(* Logix 5000 project; controller GEA_Test_Chamber vendor 1 type 14 code 196 rev 32.14; software revision 32.04; part 7 of 11 *)
(* tags used below, declared in another part *)
   FVIR_1_S_Step : INT;
   FVIR_1_W_Step : INT;
   FVIR_2_S_Step : INT;
   FVIR_2_W_Step : INT;
   FVIR_3_S_Step : INT;
   FVIR_3_W_Step : INT;
   FVIR_4_S_Step : INT;
   FVIR_4_W_Step : INT;
   FVIR_LabView_Comm_OK : BOOL;
   Start_Manequinn_Seq : BOOL;
   Start_Spill_Gasoline : BOOL;
   Start_Water_Flow_T1S : BOOL;
   Start_Water_Flow_T1W : BOOL;
   Start_Water_Flow_T2S : BOOL;
   Start_Water_Flow_T2W : BOOL;
   Start_Water_Flow_T3S : BOOL;
   Start_Water_Flow_T3W : BOOL;
   Start_Water_Flow_T4S : BOOL;
   Start_Water_Flow_T4W : BOOL;
   test : BOOL;
   Timer_Delay : TIMER[30];
   FVIR_LabView_Control : INT;
   FVIR_Test_No : INT;
   Output_FVIR : Output_FVIR;
   SET_0 : BOOL;
(* FVIR_Chamber, continued *)

ROUTINE FVIR_Test_1_Summer   (* ladder *)
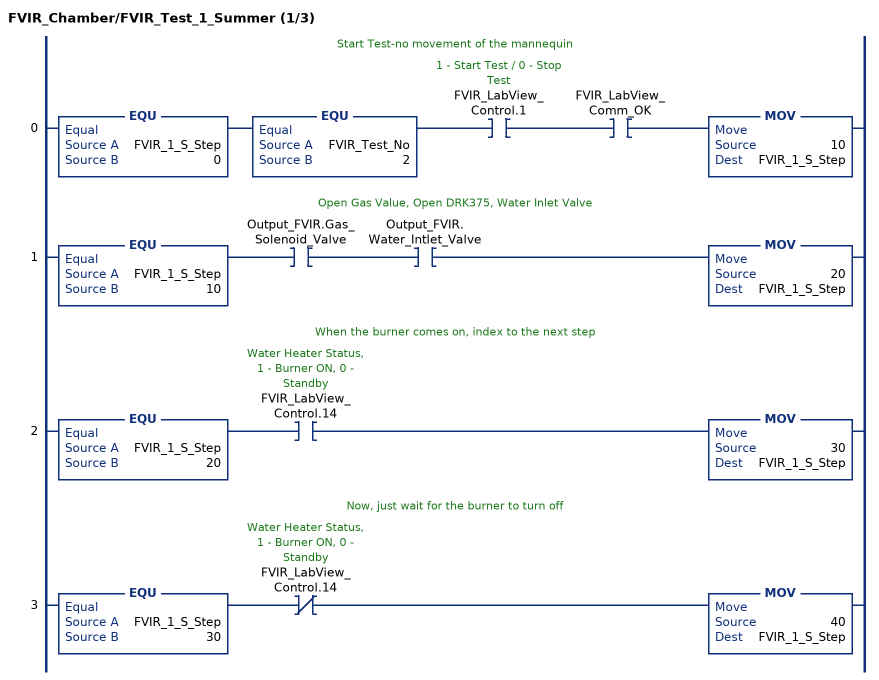
   // Start Test-no movement of the mannequin
   0: EQU(FVIR_1_S_Step,0)EQU(FVIR_Test_No,2)XIC(FVIR_LabView_Control.1)XIC(FVIR_LabView_Comm_OK)MOV(10,FVIR_1_S_Step);
   // Open Gas Value, Open DRK375, Water Inlet Valve
   1: EQU(FVIR_1_S_Step,10)XIC(Output_FVIR.Gas_Solenoid_Valve)XIC(Output_FVIR.Water_Intlet_Valve)MOV(20,FVIR_1_S_Step);
   // When the burner comes on, index to the next step
   2: EQU(FVIR_1_S_Step,20)XIC(FVIR_LabView_Control.14)MOV(30,FVIR_1_S_Step);
   // Now, just wait for the burner to turn off
   3: EQU(FVIR_1_S_Step,30)XIO(FVIR_LabView_Control.14)MOV(40,FVIR_1_S_Step);
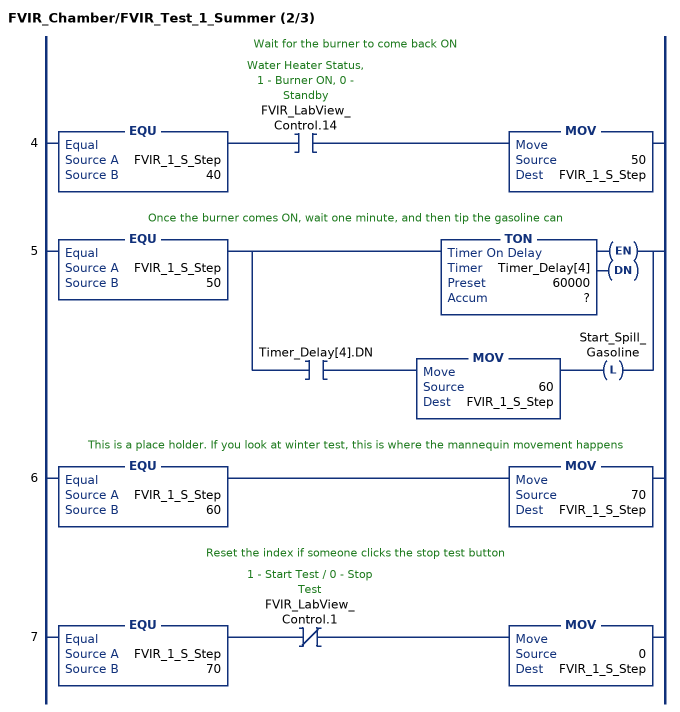
   // Wait for the burner to come back ON
   4: EQU(FVIR_1_S_Step,40)XIC(FVIR_LabView_Control.14)MOV(50,FVIR_1_S_Step);
   // Once the burner comes ON, wait one minute, and then tip the gasoline can
   5: EQU(FVIR_1_S_Step,50)[TON(Timer_Delay[4],?,?) ,XIC(Timer_Delay[4].DN) MOV(60,FVIR_1_S_Step) OTL(Start_Spill_Gasoline) ];
   // This is a place holder. If you look at winter test, this is where the mannequin movement happens
   6: EQU(FVIR_1_S_Step,60)MOV(70,FVIR_1_S_Step);
   // Reset the index if someone clicks the stop test button
   7: EQU(FVIR_1_S_Step,70)XIO(FVIR_LabView_Control.1)MOV(0,FVIR_1_S_Step);
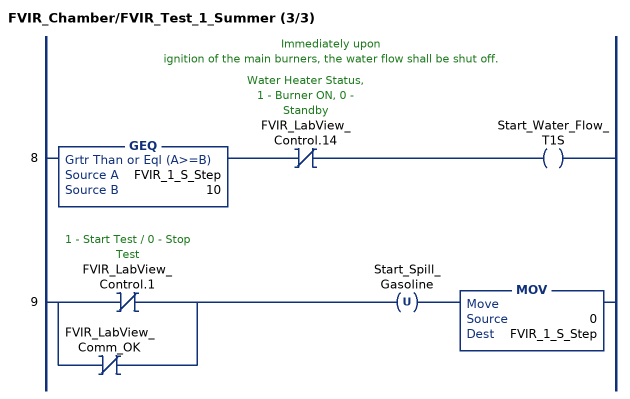
   // Immediately upon
   // ignition of the main burners, the water flow shall be shut off.
   8: GEQ(FVIR_1_S_Step,10)XIO(FVIR_LabView_Control.14)OTE(Start_Water_Flow_T1S);
   9: [XIO(FVIR_LabView_Control.1) ,XIO(FVIR_LabView_Comm_OK) ]OTU(Start_Spill_Gasoline)MOV(0,FVIR_1_S_Step);
END_ROUTINE

ROUTINE FVIR_Test_1_Winter   (* ladder *)
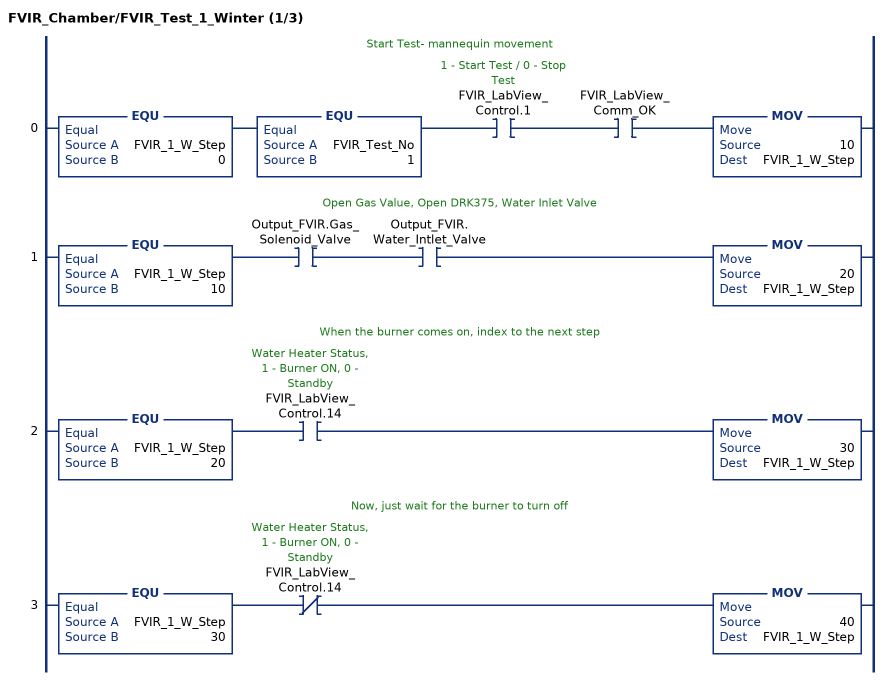
   // Start Test- mannequin movement
   0: EQU(FVIR_1_W_Step,0)EQU(FVIR_Test_No,1)XIC(FVIR_LabView_Control.1)XIC(FVIR_LabView_Comm_OK)MOV(10,FVIR_1_W_Step);
   // Open Gas Value, Open DRK375, Water Inlet Valve
   1: EQU(FVIR_1_W_Step,10)XIC(Output_FVIR.Gas_Solenoid_Valve)XIC(Output_FVIR.Water_Intlet_Valve)MOV(20,FVIR_1_W_Step);
   // When the burner comes on, index to the next step
   2: EQU(FVIR_1_W_Step,20)XIC(FVIR_LabView_Control.14)MOV(30,FVIR_1_W_Step);
   // Now, just wait for the burner to turn off
   3: EQU(FVIR_1_W_Step,30)XIO(FVIR_LabView_Control.14)MOV(40,FVIR_1_W_Step);
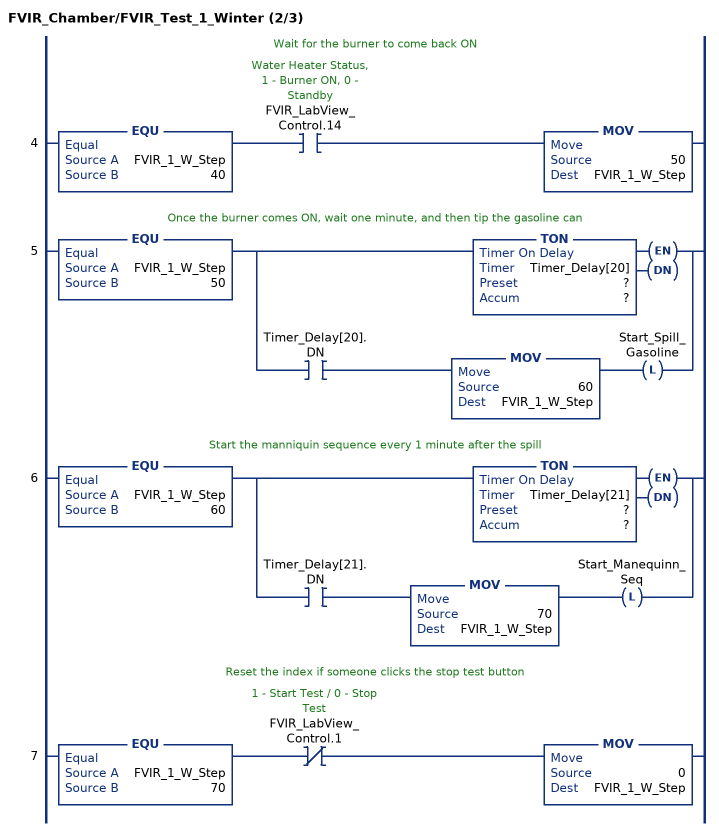
   // Wait for the burner to come back ON
   4: EQU(FVIR_1_W_Step,40)XIC(FVIR_LabView_Control.14)MOV(50,FVIR_1_W_Step);
   // Once the burner comes ON, wait one minute, and then tip the gasoline can
   5: EQU(FVIR_1_W_Step,50)[TON(Timer_Delay[20],?,?) ,XIC(Timer_Delay[20].DN) MOV(60,FVIR_1_W_Step) OTL(Start_Spill_Gasoline) ];
   // Start the manniquin sequence every 1 minute after the spill
   6: EQU(FVIR_1_W_Step,60)[TON(Timer_Delay[21],?,?) ,XIC(Timer_Delay[21].DN) MOV(70,FVIR_1_W_Step) OTL(Start_Manequinn_Seq) ];
   // Reset the index if someone clicks the stop test button
   7: EQU(FVIR_1_W_Step,70)XIO(FVIR_LabView_Control.1)MOV(0,FVIR_1_W_Step);
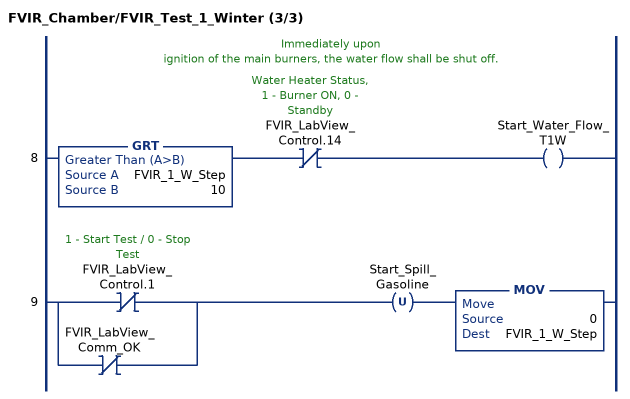
   // Immediately upon
   // ignition of the main burners, the water flow shall be shut off.
   8: GRT(FVIR_1_W_Step,10)XIO(FVIR_LabView_Control.14)OTE(Start_Water_Flow_T1W);
   9: [XIO(FVIR_LabView_Control.1) ,XIO(FVIR_LabView_Comm_OK) ]OTU(Start_Spill_Gasoline)MOV(0,FVIR_1_W_Step);
END_ROUTINE

ROUTINE FVIR_Test_2_Summer   (* ladder *)
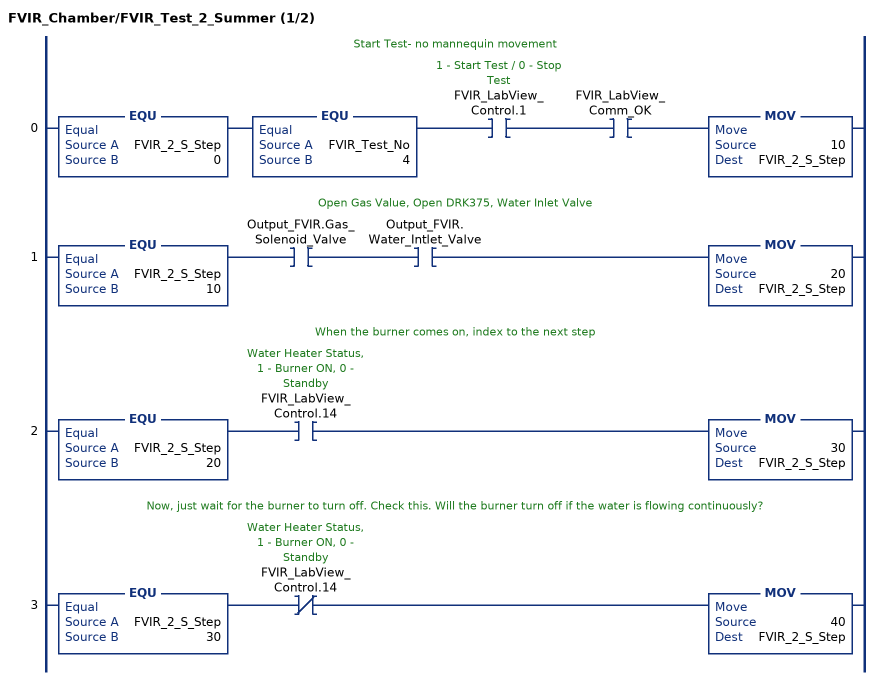
   // Start Test- no mannequin movement
   0: EQU(FVIR_2_S_Step,0)EQU(FVIR_Test_No,4)XIC(FVIR_LabView_Control.1)XIC(FVIR_LabView_Comm_OK)MOV(10,FVIR_2_S_Step);
   // Open Gas Value, Open DRK375, Water Inlet Valve
   1: EQU(FVIR_2_S_Step,10)XIC(Output_FVIR.Gas_Solenoid_Valve)XIC(Output_FVIR.Water_Intlet_Valve)MOV(20,FVIR_2_S_Step);
   // When the burner comes on, index to the next step
   2: EQU(FVIR_2_S_Step,20)XIC(FVIR_LabView_Control.14)MOV(30,FVIR_2_S_Step);
   // Now, just wait for the burner to turn off. Check this. Will the burner turn off if the water is flowing continuously?
   3: EQU(FVIR_2_S_Step,30)XIO(FVIR_LabView_Control.14)MOV(40,FVIR_2_S_Step);
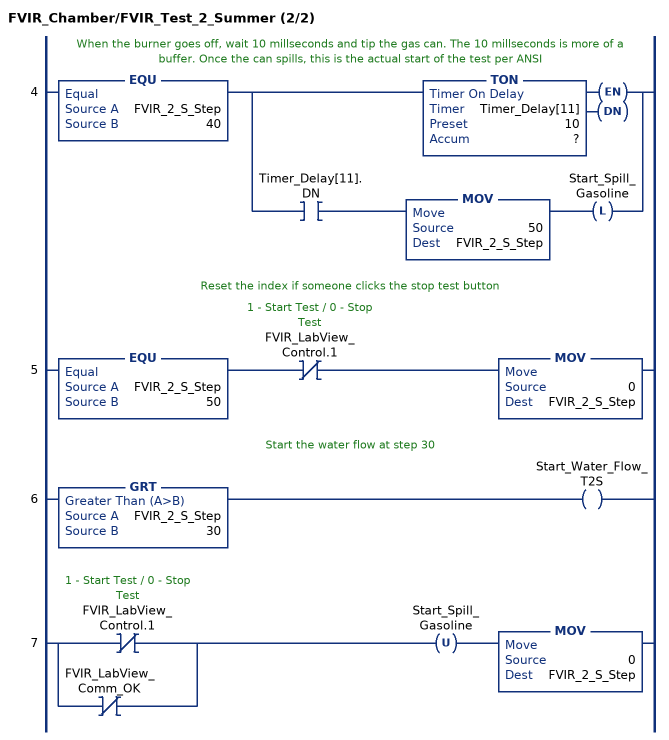
   // When the burner goes off, wait 10 millseconds and tip the gas can. The 10 millseconds is more of a buffer. Once the can spills, this is the actual start of the test per ANSI
   4: EQU(FVIR_2_S_Step,40)[TON(Timer_Delay[11],?,?) ,XIC(Timer_Delay[11].DN) MOV(50,FVIR_2_S_Step) OTL(Start_Spill_Gasoline) ];
   // Reset the index if someone clicks the stop test button
   5: EQU(FVIR_2_S_Step,50)XIO(FVIR_LabView_Control.1)MOV(0,FVIR_2_S_Step);
   // Start the water flow at step 30
   6: GRT(FVIR_2_S_Step,30)OTE(Start_Water_Flow_T2S);
   7: [XIO(FVIR_LabView_Control.1) ,XIO(FVIR_LabView_Comm_OK) ]OTU(Start_Spill_Gasoline)MOV(0,FVIR_2_S_Step);
END_ROUTINE

ROUTINE FVIR_Test_2_Winter   (* ladder *)
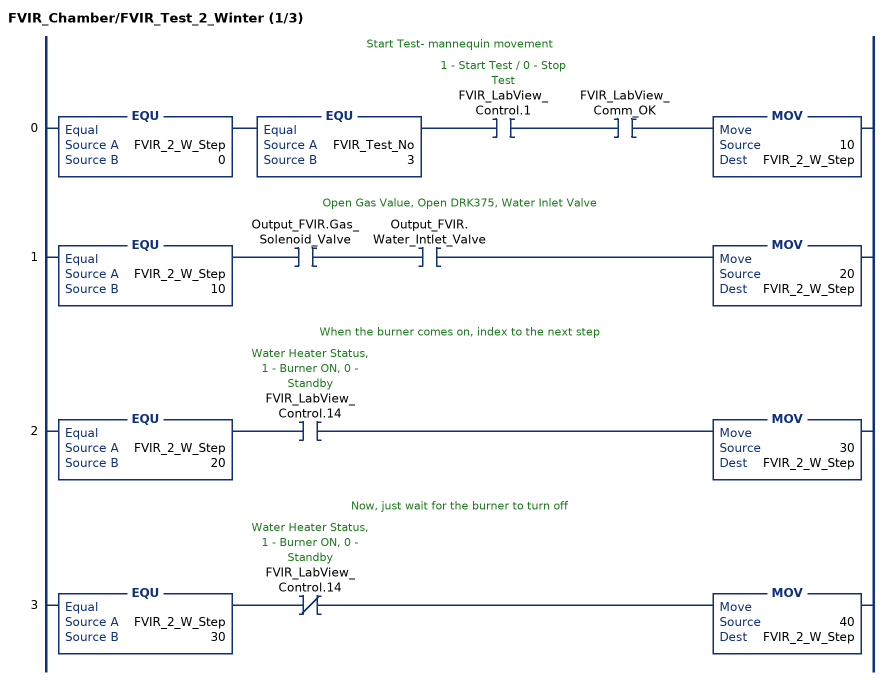
   // Start Test- mannequin movement
   0: EQU(FVIR_2_W_Step,0)EQU(FVIR_Test_No,3)XIC(FVIR_LabView_Control.1)XIC(FVIR_LabView_Comm_OK)MOV(10,FVIR_2_W_Step);
   // Open Gas Value, Open DRK375, Water Inlet Valve
   1: EQU(FVIR_2_W_Step,10)XIC(Output_FVIR.Gas_Solenoid_Valve)XIC(Output_FVIR.Water_Intlet_Valve)MOV(20,FVIR_2_W_Step);
   // When the burner comes on, index to the next step
   2: EQU(FVIR_2_W_Step,20)XIC(FVIR_LabView_Control.14)MOV(30,FVIR_2_W_Step);
   // Now, just wait for the burner to turn off
   3: EQU(FVIR_2_W_Step,30)XIO(FVIR_LabView_Control.14)MOV(40,FVIR_2_W_Step);
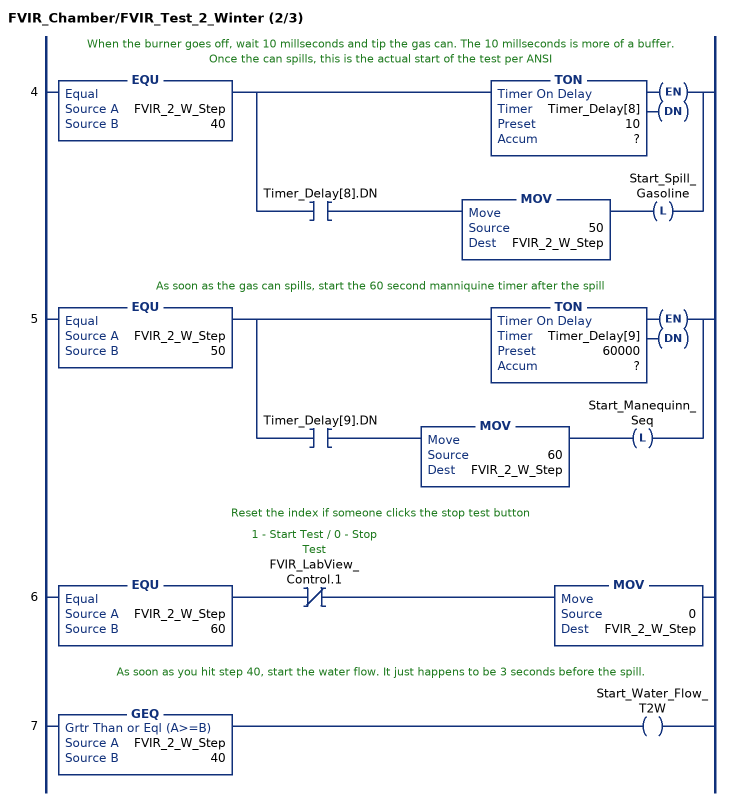
   // When the burner goes off, wait 10 millseconds and tip the gas can. The 10 millseconds is more of a buffer. Once the can spills, this is the actual start of the test per ANSI
   4: EQU(FVIR_2_W_Step,40)[TON(Timer_Delay[8],?,?) ,XIC(Timer_Delay[8].DN) MOV(50,FVIR_2_W_Step) OTL(Start_Spill_Gasoline) ];
   // As soon as the gas can spills, start the 60 second manniquine timer after the spill
   5: EQU(FVIR_2_W_Step,50)[TON(Timer_Delay[9],?,?) ,XIC(Timer_Delay[9].DN) MOV(60,FVIR_2_W_Step) OTL(Start_Manequinn_Seq) ];
   // Reset the index if someone clicks the stop test button
   6: EQU(FVIR_2_W_Step,60)XIO(FVIR_LabView_Control.1)MOV(0,FVIR_2_W_Step);
   // As soon as you hit step 40, start the water flow. It just happens to be 3 seconds before the spill.
   7: GEQ(FVIR_2_W_Step,40)OTE(Start_Water_Flow_T2W);
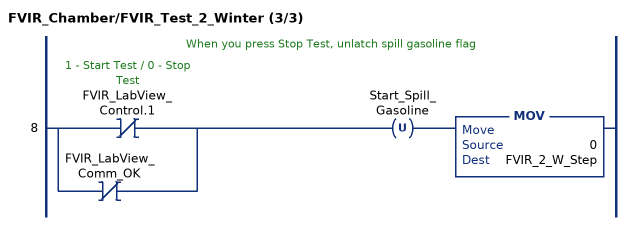
   // When you press Stop Test, unlatch spill gasoline flag
   8: [XIO(FVIR_LabView_Control.1) ,XIO(FVIR_LabView_Comm_OK) ]OTU(Start_Spill_Gasoline)MOV(0,FVIR_2_W_Step);
END_ROUTINE

ROUTINE FVIR_Test_3_Summer   (* ladder *)
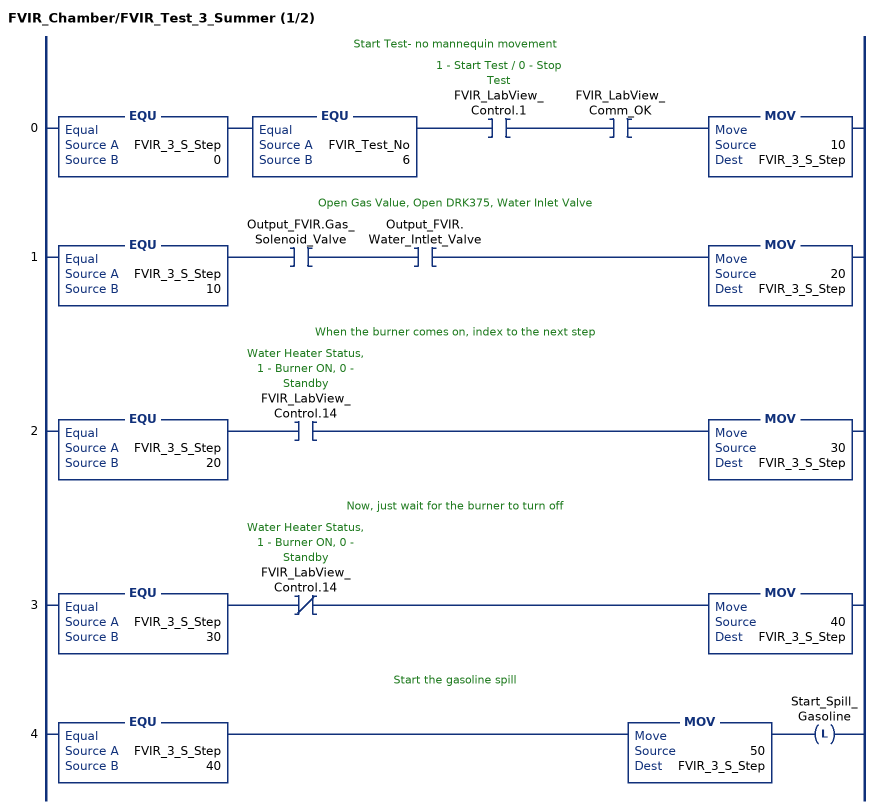
   // Start Test- no mannequin movement
   0: EQU(FVIR_3_S_Step,0)EQU(FVIR_Test_No,6)XIC(FVIR_LabView_Control.1)XIC(FVIR_LabView_Comm_OK)MOV(10,FVIR_3_S_Step);
   // Open Gas Value, Open DRK375, Water Inlet Valve
   1: EQU(FVIR_3_S_Step,10)XIC(Output_FVIR.Gas_Solenoid_Valve)XIC(Output_FVIR.Water_Intlet_Valve)MOV(20,FVIR_3_S_Step);
   // When the burner comes on, index to the next step
   2: EQU(FVIR_3_S_Step,20)XIC(FVIR_LabView_Control.14)MOV(30,FVIR_3_S_Step);
   // Now, just wait for the burner to turn off
   3: EQU(FVIR_3_S_Step,30)XIO(FVIR_LabView_Control.14)MOV(40,FVIR_3_S_Step);
   // Start the gasoline spill
   4: EQU(FVIR_3_S_Step,40)MOV(50,FVIR_3_S_Step)OTL(Start_Spill_Gasoline);
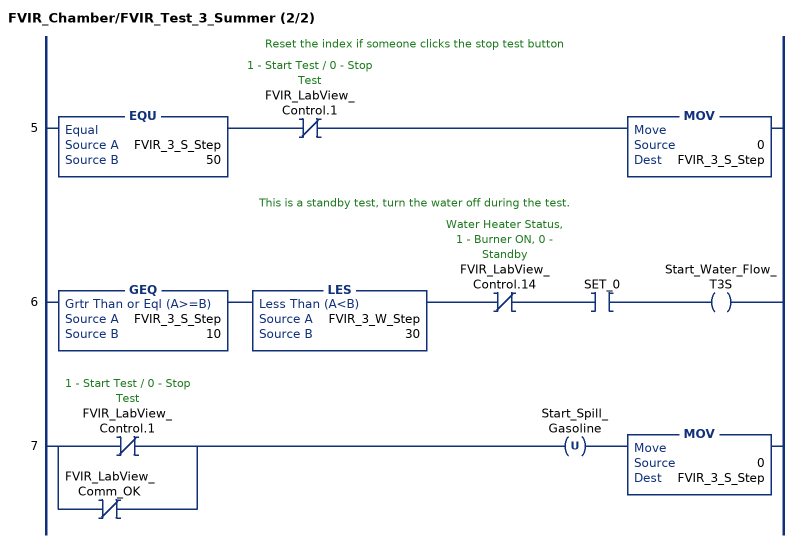
   // Reset the index if someone clicks the stop test button
   5: EQU(FVIR_3_S_Step,50)XIO(FVIR_LabView_Control.1)MOV(0,FVIR_3_S_Step);
   // This is a standby test, turn the water off during the test.
   6: GEQ(FVIR_3_S_Step,10)LES(FVIR_3_W_Step,30)XIO(FVIR_LabView_Control.14)XIC(SET_0)OTE(Start_Water_Flow_T3S);
   7: [XIO(FVIR_LabView_Control.1) ,XIO(FVIR_LabView_Comm_OK) ]OTU(Start_Spill_Gasoline)MOV(0,FVIR_3_S_Step);
END_ROUTINE

ROUTINE FVIR_Test_3_Winter   (* ladder *)
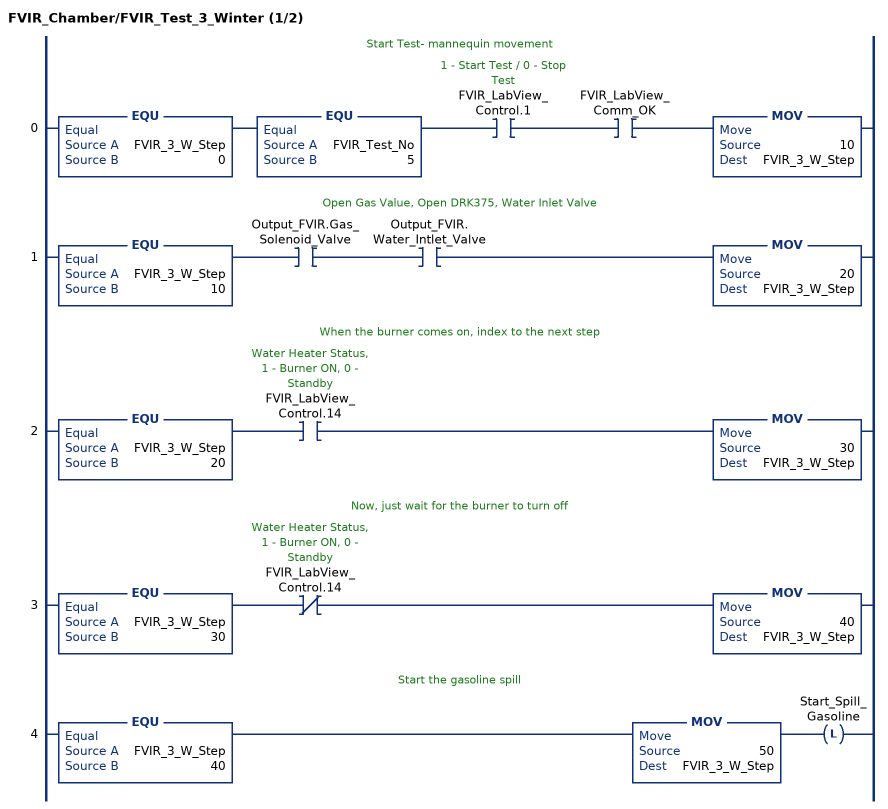
   // Start Test- mannequin movement
   0: EQU(FVIR_3_W_Step,0)EQU(FVIR_Test_No,5)XIC(FVIR_LabView_Control.1)XIC(FVIR_LabView_Comm_OK)MOV(10,FVIR_3_W_Step);
   // Open Gas Value, Open DRK375, Water Inlet Valve
   1: EQU(FVIR_3_W_Step,10)XIC(Output_FVIR.Gas_Solenoid_Valve)XIC(Output_FVIR.Water_Intlet_Valve)MOV(20,FVIR_3_W_Step);
   // When the burner comes on, index to the next step
   2: EQU(FVIR_3_W_Step,20)XIC(FVIR_LabView_Control.14)MOV(30,FVIR_3_W_Step);
   // Now, just wait for the burner to turn off
   3: EQU(FVIR_3_W_Step,30)XIO(FVIR_LabView_Control.14)MOV(40,FVIR_3_W_Step);
   // Start the gasoline spill
   4: EQU(FVIR_3_W_Step,40)MOV(50,FVIR_3_W_Step)OTL(Start_Spill_Gasoline);
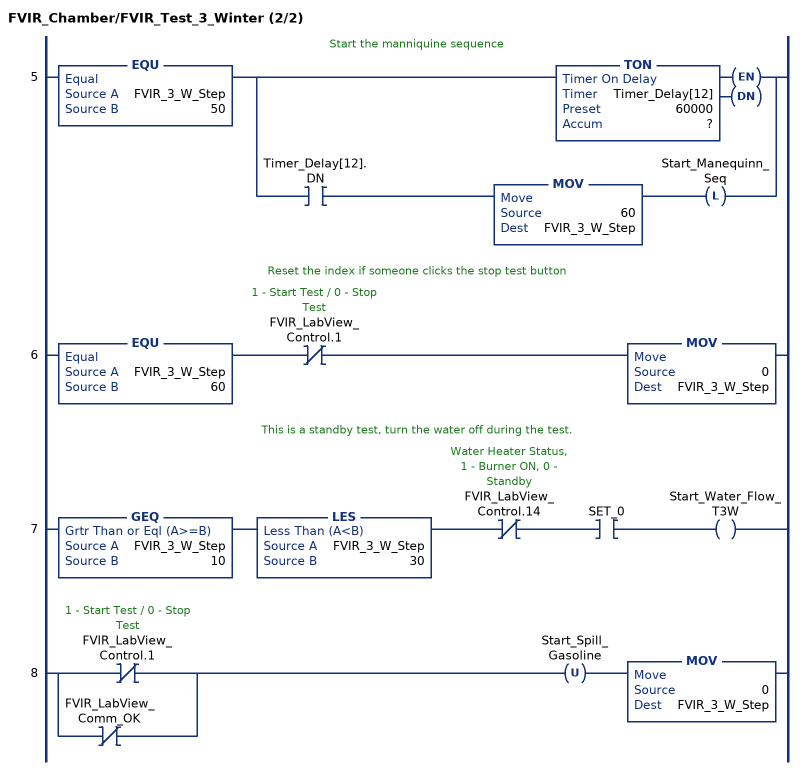
   // Start the manniquine sequence
   5: EQU(FVIR_3_W_Step,50)[TON(Timer_Delay[12],?,?) ,XIC(Timer_Delay[12].DN) MOV(60,FVIR_3_W_Step) OTL(Start_Manequinn_Seq) ];
   // Reset the index if someone clicks the stop test button
   6: EQU(FVIR_3_W_Step,60)XIO(FVIR_LabView_Control.1)MOV(0,FVIR_3_W_Step);
   // This is a standby test, turn the water off during the test.
   7: GEQ(FVIR_3_W_Step,10)LES(FVIR_3_W_Step,30)XIO(FVIR_LabView_Control.14)XIC(SET_0)OTE(Start_Water_Flow_T3W);
   8: [XIO(FVIR_LabView_Control.1) ,XIO(FVIR_LabView_Comm_OK) ]OTU(Start_Spill_Gasoline)MOV(0,FVIR_3_W_Step);
END_ROUTINE

ROUTINE FVIR_Test_4_Summer   (* ladder *)
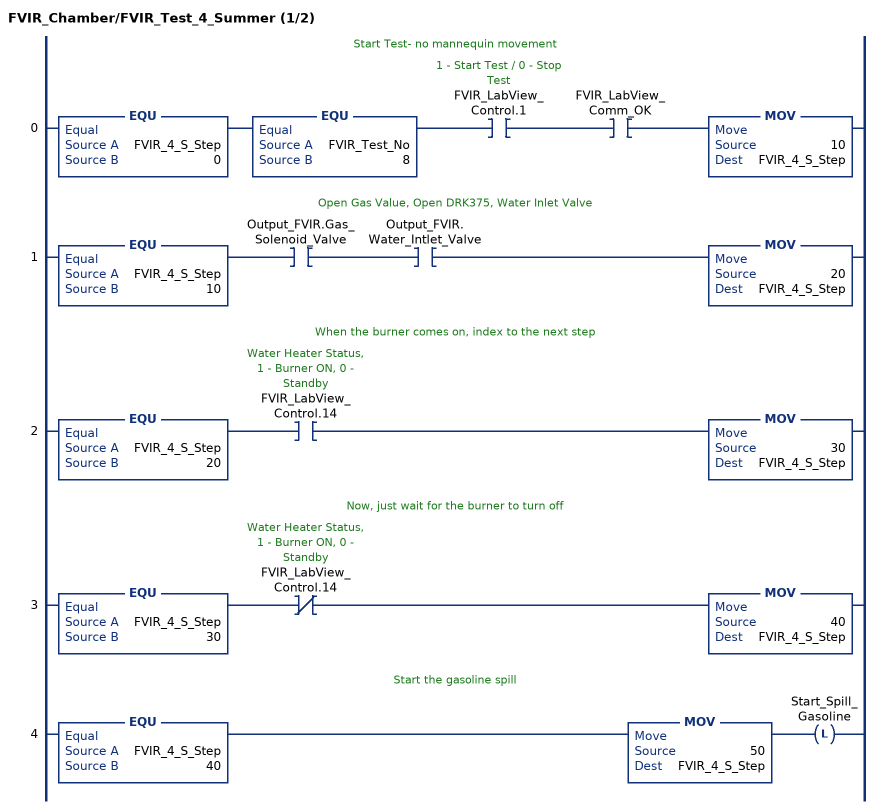
   // Start Test- no mannequin movement
   0: EQU(FVIR_4_S_Step,0)EQU(FVIR_Test_No,8)XIC(FVIR_LabView_Control.1)XIC(FVIR_LabView_Comm_OK)MOV(10,FVIR_4_S_Step);
   // Open Gas Value, Open DRK375, Water Inlet Valve
   1: EQU(FVIR_4_S_Step,10)XIC(Output_FVIR.Gas_Solenoid_Valve)XIC(Output_FVIR.Water_Intlet_Valve)MOV(20,FVIR_4_S_Step);
   // When the burner comes on, index to the next step
   2: EQU(FVIR_4_S_Step,20)XIC(FVIR_LabView_Control.14)MOV(30,FVIR_4_S_Step);
   // Now, just wait for the burner to turn off
   3: EQU(FVIR_4_S_Step,30)XIO(FVIR_LabView_Control.14)MOV(40,FVIR_4_S_Step);
   // Start the gasoline spill
   4: EQU(FVIR_4_S_Step,40)MOV(50,FVIR_4_S_Step)OTL(Start_Spill_Gasoline);
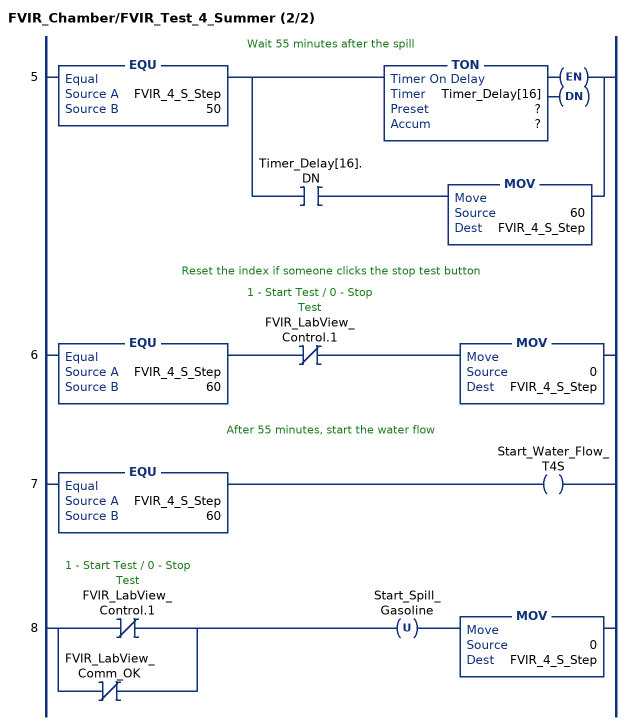
   // Wait 55 minutes after the spill
   5: EQU(FVIR_4_S_Step,50)[TON(Timer_Delay[16],?,?) ,XIC(Timer_Delay[16].DN) MOV(60,FVIR_4_S_Step) ];
   // Reset the index if someone clicks the stop test button
   6: EQU(FVIR_4_S_Step,60)XIO(FVIR_LabView_Control.1)MOV(0,FVIR_4_S_Step);
   // After 55 minutes, start the water flow
   7: EQU(FVIR_4_S_Step,60)OTE(Start_Water_Flow_T4S);
   8: [XIO(FVIR_LabView_Control.1) ,XIO(FVIR_LabView_Comm_OK) ]OTU(Start_Spill_Gasoline)MOV(0,FVIR_4_S_Step);
END_ROUTINE

ROUTINE FVIR_Test_4_Winter   (* ladder *)
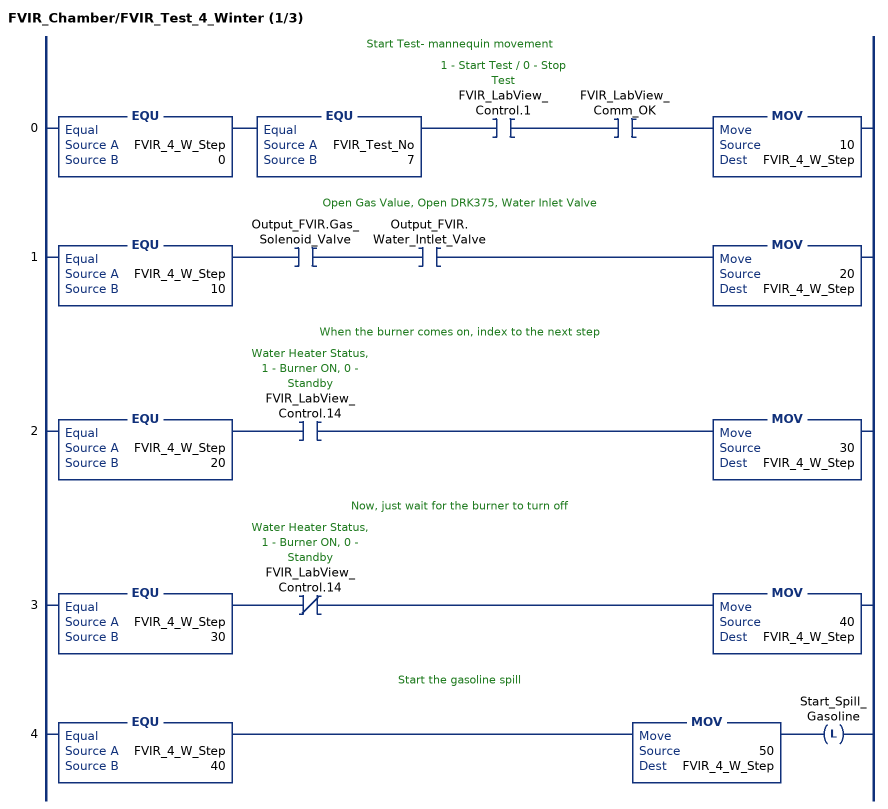
   // Start Test- mannequin movement
   0: EQU(FVIR_4_W_Step,0)EQU(FVIR_Test_No,7)XIC(FVIR_LabView_Control.1)XIC(FVIR_LabView_Comm_OK)MOV(10,FVIR_4_W_Step);
   // Open Gas Value, Open DRK375, Water Inlet Valve
   1: EQU(FVIR_4_W_Step,10)XIC(Output_FVIR.Gas_Solenoid_Valve)XIC(Output_FVIR.Water_Intlet_Valve)MOV(20,FVIR_4_W_Step);
   // When the burner comes on, index to the next step
   2: EQU(FVIR_4_W_Step,20)XIC(FVIR_LabView_Control.14)MOV(30,FVIR_4_W_Step);
   // Now, just wait for the burner to turn off
   3: EQU(FVIR_4_W_Step,30)XIO(FVIR_LabView_Control.14)MOV(40,FVIR_4_W_Step);
   // Start the gasoline spill
   4: EQU(FVIR_4_W_Step,40)MOV(50,FVIR_4_W_Step)OTL(Start_Spill_Gasoline);
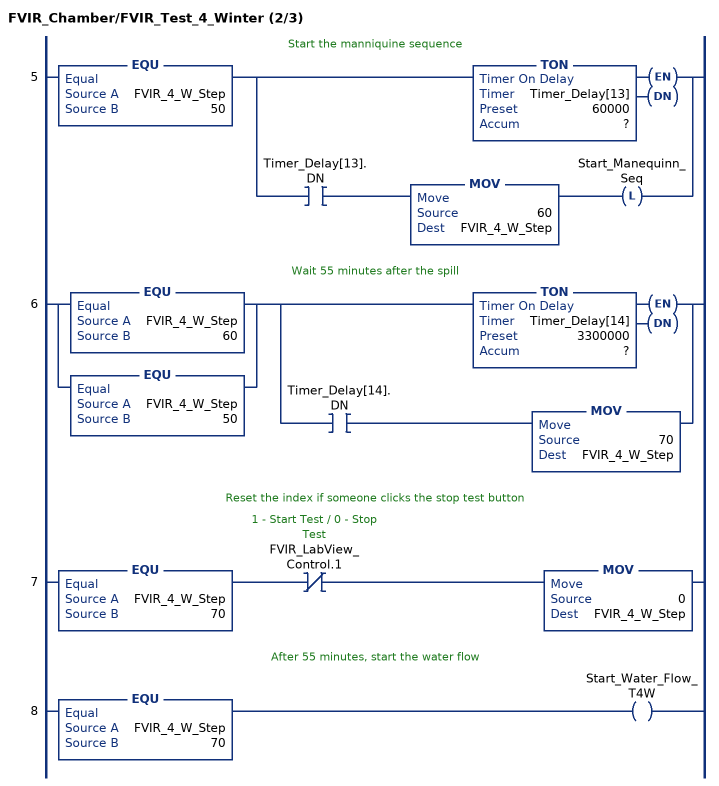
   // Start the manniquine sequence
   5: EQU(FVIR_4_W_Step,50)[TON(Timer_Delay[13],?,?) ,XIC(Timer_Delay[13].DN) MOV(60,FVIR_4_W_Step) OTL(Start_Manequinn_Seq) ];
   // Wait 55 minutes after the spill
   6: [EQU(FVIR_4_W_Step,60) ,EQU(FVIR_4_W_Step,50) ][TON(Timer_Delay[14],?,?) ,XIC(Timer_Delay[14].DN) MOV(70,FVIR_4_W_Step) ];
   // Reset the index if someone clicks the stop test button
   7: EQU(FVIR_4_W_Step,70)XIO(FVIR_LabView_Control.1)MOV(0,FVIR_4_W_Step);
   // After 55 minutes, start the water flow
   8: EQU(FVIR_4_W_Step,70)OTE(Start_Water_Flow_T4W);
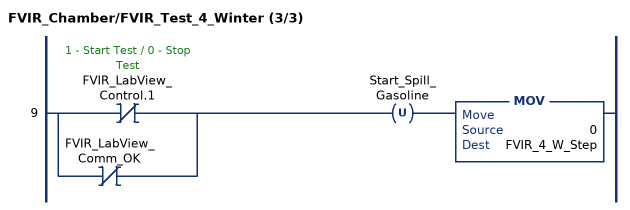
   9: [XIO(FVIR_LabView_Control.1) ,XIO(FVIR_LabView_Comm_OK) ]OTU(Start_Spill_Gasoline)MOV(0,FVIR_4_W_Step);
END_ROUTINE
END_PROGRAM
